// Implicitly generated code : DO NOT EDIT
FUNCTION CheckRangeSigned : DINT
VAR_INPUT
	value, lower, upper: DINT;
END_VAR

// Implicitly generated code : Only an Implementation suggestion
{noflow}
IF (value < lower) THEN
	CheckRangeSigned := lower;
ELSIF(value > upper) THEN
	CheckRangeSigned := upper;
ELSE
	CheckRangeSigned := value;
END_IF
{flow}

END_FUNCTION

(* stored: Version 1.1.0.1, ProductVersion 3.1.4024.2
   POU CheckRangeSigned: Id {ff7a1b9d-b4bf-4f88-a085-e8fe451f8e6c}, SpecialFunc CheckRangeSigned *)
